{attribute addProperty _moveHomeDefaultName "<#MOVE HOME#>"}
{attribute addProperty _moveWorkDefaultName "<#MOVE TO WORK#>"}
{attribute addProperty _stopDefaultName "<#STOP#>"}
FUNCTION_BLOCK TcoCylinder EXTENDS TcoCylinderBase
VAR
    {attribute addProperty Name "|[[1]Attribute_moveHomeDefaultName]|"}
    _moveHomeDefault : TcoCylinderMoveTask(THIS^);
    {attribute addProperty Name "|[[1]Attribute_moveWorkDefaultName]|"}
    _moveWorkDefault : TcoCylinderMoveTask(THIS^);
    {attribute addProperty Name "|[[1]Attribute_stopDefaultName]|"}
    _stopDefault : TcoCore.TcoTask(THIS^);
	increment: INT;
	_suspendedHome:BOOL;
	_suspendedWork:BOOL;
	{attribute 'hide'} 
	_suspendedHomeCounter:INT;
	{attribute 'hide'} 
	_suspendedWorkCounter:INT;
END_VAR
VAR
    _config : TcoCylinderConfig;
	_status : TcoCylinderStatus;
	_refillTimer:TON;	
END_VAR

SUPER^(inoAtHomePos := inoAtHomePos, inoAtWorkPos := inoAtWorkPos, inoToHomePos := inoToHomePos, inoToWorkPos := inoToWorkPos);
_suspendedHomeCounter:=0;
_suspendedWorkCounter:=0;

	
IF(_atHomePos AND _atWorkPos) THEN Messenger.Error('<#Home and work position sensors are both active. Check the position of sensors!#>'); END_IF;

// Disables mutualy exclusive actions
_moveWorkDefault.Enabled := TRUE;// NOT _moveHomeDefault.Busy;


_moveHomeDefault(PositionSensor := _atHomePos AND NOT _atWorkPos,
    MoveToPositionSignal := _toHomePos,
    InverseSignal := _toWorkPos,
	TimeToRefill:=_config.TimeToRefill,
	refInverseTask:=_moveWorkDefault,
    MaxTimeToReachPosition := _config.TimeToReachHomePosition,
    PositionName := '<#Home#>');


	
// Disables mutualy exclusive actions		
_moveHomeDefault.Enabled := TRUE;//NOT _moveWorkDefault.Busy;
	
_moveWorkDefault(PositionSensor := _atWorkPos AND NOT _atHomePos,
    MoveToPositionSignal := _toWorkPos,
    InverseSignal := _toHomePos,
	TimeToRefill:=_config.TimeToRefill,
	refInverseTask:=_moveHomeDefault,
    MaxTimeToReachPosition := _config.TimeToReachWorkPosition,
    PositionName := '<#Work#>');
	

IF (_stopDefault.Execute()) THEN
	_toHomePos := FALSE;
	_toWorkPos := FALSE;
    _moveHomeDefault.Abort();
    _moveWorkDefault.Abort();
    _stopDefault.Abort();
    _moveHomeDefault.Restore();
    _moveWorkDefault.Restore();
    _stopDefault.Restore();
    _stopDefault.DoneWhen(TRUE);
END_IF



// For further discussion about Status
IF(_moveHomeDefault.Busy) THEN
	_status.ActionDescription := 'Moving to home position';
ELSIF(_moveWorkDefault.Busy) THEN
	_status.ActionDescription := 'Moving to work position';
ELSIF(_stopDefault.Busy) THEN
	_status.ActionDescription := 'Stopping pressure';
ELSE	
	_status.ActionDescription := 'Idle';
END_IF

SUPER^(inoAtHomePos := inoAtHomePos, inoAtWorkPos := inoAtWorkPos, inoToHomePos := inoToHomePos, inoToWorkPos := inoToWorkPos);

(*~
	<docu>
		<summary>
			Aborts the movement to home position when the condition is 'true'.
		</summary>
		<remarks>			
				<note type="warning">
					The call of this method will be effective only when called AFTER the initialization of the instance of given TcoCylinder.
				</note>
		</remarks>	
	</docu>
~*)
METHOD AbortMoveHome : BOOL
VAR_IN_OUT
	(*~
	<docu>
		<summary>
			Condition to abort the movement of the cylinder.
		</summary>	
	</docu>
	~*)
	inoDisableCondition : BOOL;
END_VAR
VAR
	_signalInfo : TcoSignalInfo;
END_VAR
IF (_toHomePos OR _moveHomeDefault.Busy) AND inoDisableCondition THEN
	_signalInfo.GetSignalInfo(SIZEOF(inoDisableCondition), ADR(inoDisableCondition));
	Messenger.Build().Append('<#Movement aborted due to#> : ').Append(_signalInfo.SymbolPath).As().AsError().Pin();
	_toHomePos := FALSE;
	IF(__ISVALIDREF(THIS^.inoToHomePos)) THEN THIS^.inoToHomePos := FALSE; END_IF;
	_moveHomeDefault.Abort();
END_IF
END_METHOD

(*~
	<docu>
		<summary>
			Aborts the movement to work position when the condition is 'true'.
		</summary>
		<remarks>			
				<note type="warning">
					The call of this method will be effective only when called AFTER the initialization of the instance of given TcoCylinder.
				</note>
		</remarks>	
	</docu>
~*)
METHOD AbortMoveWork : BOOL
VAR_IN_OUT
	(*~
		<docu>
			<summary>
				Condition to abort the movement of the cylinder.
			</summary>	
		</docu>
	~*)
	inoDisableCondition : BOOL;
END_VAR
VAR
	_signalInfo : TcoSignalInfo;
END_VAR
IF (_toWorkPos OR _moveWorkDefault.Busy) AND inoDisableCondition THEN
	_signalInfo.GetSignalInfo(SIZEOF(inoDisableCondition), ADR(inoDisableCondition));
	Messenger.Build().Append('<#Movement aborted due to#> : ').Append(_signalInfo.SymbolPath).As().AsError().Pin();
	_toWorkPos := FALSE;
	IF(__ISVALIDREF(THIS^.inoToWorkPos)) THEN THIS^.inoToWorkPos := FALSE; END_IF;
	_moveWorkDefault.Abort();
END_IF
END_METHOD

(*~
	<docu>
		<summary>
			Gets the configuration of the cylinder. 					
		</summary>			
	</docu>	
~*)
PROPERTY Config : REFERENCE TO TcoCylinderConfig
GET
Config REF= _config;
END_GET
END_PROPERTY

(*~
	<docu>
		<summary>
			Gets the `MoveHomeTask` task that controls the moving of the cyclinder in home position. 		
		</summary>			
	</docu>	
~*)
PROPERTY MoveHomeTask : TcoCore.ITcoTask
GET
MoveHomeTask := _moveHomeDefault;
END_GET
END_PROPERTY

(*~
	<docu>
		<summary>
			Gets the `MoveWorkTask` task that controls the moving of the cyclinder into work position. 		
		</summary>			
	</docu>	
~*)
PROPERTY MoveWorkTask : TcoCore.ITcoTask
GET
MoveWorkTask := _moveWorkDefault;
END_GET
END_PROPERTY

(*~
	<docu>
		<summary>
			Refill cylinder after booth outputs are off .
		</summary>
		<remarks>			
				<note type="warning">
					The call of this method will be effective only when called AFTER the initialization of the instance of given TcoCylinder and methods like AbortMoveHone,SuspendMoveHom...
				</note>
		</remarks>	
	</docu>
~*)
METHOD Refill : BOOL
VAR_INPUT
	(*~
	<docu>
		<summary>
			Time of refill cylinder after aborting or suspending
		</summary>	
	</docu>
	~*)
	inRefillTime:TIME;
END_VAR

_refillTimer(In:=inoToHomePos XOR  inoToWorkPos ,Pt:=T#49D);

_config.TimeToRefill:=inRefillTime;

IF  _refillTimer.ET>T#0MS
	AND _refillTimer.ET<_config.TimeToRefill  
	AND _config.TimeToRefill<>T#0S THEN
	_toHomePos	 := TRUE;
	_toWorkPos	 := TRUE;	
END_IF;

	
SUPER^(inoAtHomePos := inoAtHomePos, inoAtWorkPos := inoAtWorkPos, inoToHomePos := inoToHomePos, inoToWorkPos := inoToWorkPos);
END_METHOD

PROPERTY Status : REFERENCE TO TcoCylinderStatus
GET
Status REF= _status;
END_GET
END_PROPERTY

(*~
	<docu>
		<summary>
			Gets the `StopTask` task that controls the stopping of the cyclinder. 		
		</summary>			
	</docu>	
~*)
PROPERTY StopTask : TcoCore.ITcoTask
GET
StopTask := _stopDefault;
END_GET
END_PROPERTY

(*~
	<docu>
		<summary>
			Suspend the movement to home position when the condition is 'true'. Task is still busy
		</summary>
		<remarks>			
				<note type="warning">
					The call of this method will be effective only when called AFTER the initialization of the instance of given TcoCylinder.
				</note>
		</remarks>	
	</docu>
~*)
METHOD SuspendMoveHome : BOOL
VAR_IN_OUT
	(*~
	<docu>
		<summary>
			Condition to abort the movement of the cylinder.
		</summary>	
	</docu>
	~*)
	inoDisableCondition : BOOL;
END_VAR
VAR
	_signalInfo : TcoSignalInfo;
END_VAR
IF inoDisableCondition THEN
	_suspendedHomeCounter:=_suspendedHomeCounter+1;
END_IF
_suspendedHome:=_suspendedHomeCounter>0;

IF (_toHomePos OR _moveHomeDefault.Busy) AND inoDisableCondition THEN
	_signalInfo.GetSignalInfo(SIZEOF(inoDisableCondition), ADR(inoDisableCondition));
	Messenger.Warning(CONCAT('<#Movement suspended due to#> : ' , _signalInfo.SymbolPath));
	_toHomePos := FALSE;
	IF(__ISVALIDREF(THIS^.inoToHomePos)) THEN THIS^.inoToHomePos := FALSE; END_IF;
	
END_IF
END_METHOD

METHOD SuspendMoveHomeExpression : BOOL
VAR_INPUT
		inDisableCondition : BOOL;
		inMessage:STRING;
END_VAR
IF inDisableCondition THEN
	_suspendedHomeCounter:=_suspendedHomeCounter+1;
END_IF
_suspendedHome:=_suspendedHomeCounter>0;

IF (_toHomePos OR _moveHomeDefault.Busy) AND inDisableCondition THEN
	Messenger.Warning(CONCAT('<#Movement suspended due to#> : ' , inMessage));
	_toHomePos := FALSE;
	IF(__ISVALIDREF(THIS^.inoToHomePos)) THEN THIS^.inoToHomePos := FALSE; END_IF;
	
END_IF;
END_METHOD

(*~
	<docu>
		<summary>
			Suspend the movement to home position when the condition is NOT 'true'. Task is still busy
		</summary>
		<remarks>			
				<note type="warning">
					The call of this method will be effective only when called AFTER the initialization of the instance of given TcoCylinder.
				</note>
		</remarks>	
	</docu>
~*)
METHOD SuspendMoveHomeInverted : BOOL
VAR_IN_OUT
	(*~
	<docu>
		<summary>
			Condition to abort the movement of the cylinder.
		</summary>	
	</docu>
	~*)
	inoDisableCondition : BOOL;
END_VAR
VAR
	_signalInfo : TcoSignalInfo;
END_VAR
IF inoDisableCondition THEN
	_suspendedHomeCounter:=_suspendedHomeCounter+1;
END_IF
_suspendedHome:=_suspendedHomeCounter>0;

IF (_toHomePos OR _moveHomeDefault.Busy) AND not inoDisableCondition THEN
	_signalInfo.GetSignalInfo(SIZEOF(inoDisableCondition), ADR(inoDisableCondition));
	Messenger.Warning(CONCAT('<#Movement suspended due to NOT#> : ' , _signalInfo.SymbolPath));
	_toHomePos := FALSE;
	IF(__ISVALIDREF(THIS^.inoToHomePos)) THEN THIS^.inoToHomePos := FALSE; END_IF;
	
END_IF
END_METHOD

(*~
	<docu>
		<summary>
			Suspend the movement to work position when the condition is 'true'. Task is still bussy
		</summary>
		<remarks>			
				<note type="warning">
					The call of this method will be effective only when called AFTER the initialization of the instance of given TcoCylinder.
				</note>
		</remarks>	
	</docu>
~*)
METHOD SuspendMoveWork : BOOL
VAR_IN_OUT
	(*~
		<docu>
			<summary>
				Condition to abort the movement of the cylinder.
			</summary>	
		</docu>
	~*)
	inoDisableCondition : BOOL;
END_VAR
VAR
	_signalInfo : TcoSignalInfo;
END_VAR
IF inoDisableCondition THEN
	_suspendedWorkCounter:=_suspendedWorkCounter+1;
END_IF
_suspendedWork:=_suspendedWorkCounter>0;

IF (_toWorkPos OR _moveWorkDefault.Busy) AND inoDisableCondition THEN
	_signalInfo.GetSignalInfo(SIZEOF(inoDisableCondition), ADR(inoDisableCondition));
	Messenger.Warning(CONCAT('<#Movement suspended due to#> : ' , _signalInfo.SymbolPath));
	_toWorkPos := FALSE;
	IF(__ISVALIDREF(THIS^.inoToWorkPos)) THEN THIS^.inoToWorkPos := FALSE; END_IF;

END_IF
END_METHOD

METHOD SuspendMoveWorkExpression : BOOL
VAR_INPUT
		inDisableCondition : BOOL;
		inMessage:STRING;
END_VAR
IF inDisableCondition THEN
	_suspendedWorkCounter:=_suspendedWorkCounter+1;
END_IF
_suspendedWork:=_suspendedWorkCounter>0;

IF (_toWorkPos OR _moveWorkDefault.Busy) AND inDisableCondition THEN
    Messenger.Warning(CONCAT('<#Movement suspended due to#> : ', inMessage));
    _toWorkPos := FALSE;
    IF (__ISVALIDREF(THIS^.inoToWorkPos)) THEN
        THIS^.inoToWorkPos := FALSE;
    END_IF;

END_IF
END_METHOD

(*~
	<docu>
		<summary>
			Suspend the movement to work position when the condition is NOT 'true'. Task is still busy
		</summary>
		<remarks>			
				<note type="warning">
					The call of this method will be effective only when called AFTER the initialization of the instance of given TcoCylinder.
				</note>
		</remarks>	
	</docu>
~*)
METHOD SuspendMoveWorkInverted : BOOL
VAR_IN_OUT
	(*~
		<docu>
			<summary>
				Condition to abort the movement of the cylinder.
			</summary>	
		</docu>
	~*)
	inoDisableCondition : BOOL;
END_VAR
VAR
	_signalInfo : TcoSignalInfo;
END_VAR
IF inoDisableCondition THEN
	_suspendedWorkCounter:=_suspendedWorkCounter+1;
END_IF
_suspendedWork:=_suspendedWorkCounter>0;

IF (_toWorkPos OR _moveWorkDefault.Busy) AND not inoDisableCondition THEN
    _signalInfo.GetSignalInfo(SIZEOF(inoDisableCondition), ADR(inoDisableCondition));
    Messenger.Warning(CONCAT('<#Movement suspended due to NOT#> : ', _signalInfo.SymbolPath));
    _toWorkPos := FALSE;
    IF (__ISVALIDREF(THIS^.inoToWorkPos)) THEN
        THIS^.inoToWorkPos := FALSE;
    END_IF;

END_IF
END_METHOD

END_FUNCTION_BLOCK

(* stored: Version 1.1.0.1, ProductVersion 3.1.4024.12
   POU TcoCylinder: Id {fe4e2550-76ec-4019-82bb-e68b2cbe4d49}, SpecialFunc None
   Folder Suspend: Id {4644ecd8-38e1-0b3a-2c11-f033423ed87b}
   Folder Tasks: Id {2c49a519-7477-00ef-0cce-12b7d5ee9e41}
   Method AbortMoveHome: Id {47e4576d-3c08-01cc-0965-20c209cad595}
   Method AbortMoveWork: Id {9c09b925-4ae8-044b-2972-72392d722888}
   Property Config: Id {4900e490-aca6-01f6-34b5-8e88d5861bd7}
   Get Get: Id {01381d79-df26-0dfc-0b34-6d73c1b5b634}
   Property MoveHomeTask: Id {6c5528f8-8b8f-0e7d-01e4-787b210fe4ca}
   Get Get: Id {5717e4b3-14ff-0743-005a-b365bdc9a2e1}
   Property MoveWorkTask: Id {b7eb0230-cd38-0ac9-3271-cda0637a6c51}
   Get Get: Id {d38ced05-e6e6-0894-2289-cb1e2f89ee7d}
   Method Refill: Id {c33ee3d5-77c3-0060-11e3-8b63ed6f8e3a}
   Property Status: Id {4e25aab9-b7e5-00e7-1126-2a4313a14d92}
   Get Get: Id {a32a112b-8373-0a19-170b-cdfdf4b5b4dd}
   Property StopTask: Id {f45f0198-4c17-0e92-3a52-5cc8984cb39c}
   Get Get: Id {28fe28be-dd9b-0922-165d-691ae597ebf9}
   Method SuspendMoveHome: Id {128f7344-e079-082c-17fd-86f14c85bfff}
   Method SuspendMoveHomeExpression: Id {509ab9da-646e-0ba9-2ee9-e45e4d652ad0}
   Method SuspendMoveHomeInverted: Id {93e3d535-9b9b-08a5-2e0f-81451efdb8a6}
   Method SuspendMoveWork: Id {f52d30db-3f57-05e7-265a-4214e83dd76b}
   Method SuspendMoveWorkExpression: Id {ceff43ee-f027-07c3-1593-7f35dabaedd3}
   Method SuspendMoveWorkInverted: Id {0a6cb00f-a9de-0384-275e-638c4f00395c} *)
